            CASE Value 
OF
  SplineMode.DISCRETE_POINTS      : SPLINE_MODE_TO_STRING := StrReplace('DISCRETE_POINTS ({0})'      ,'{0}' , UINT_TO_STRING(Value));
  SplineMode.BEZIER_SPLINE        : SPLINE_MODE_TO_STRING := StrReplace('BEZIER_SPLINE ({0})'        ,'{0}' , UINT_TO_STRING(Value));
  SplineMode.B_SPLINES            : SPLINE_MODE_TO_STRING := StrReplace('B_SPLINES ({0})'            ,'{0}' , UINT_TO_STRING(Value));
  SplineMode.CUBIC_HERMITE_SPLINE : SPLINE_MODE_TO_STRING := StrReplace('CUBIC_HERMITE_SPLINE ({0})' ,'{0}' , UINT_TO_STRING(Value));
  SplineMode.C_SPLINES            : SPLINE_MODE_TO_STRING := StrReplace('C_SPLINES ({0})'            ,'{0}' , UINT_TO_STRING(Value));
ELSE
  SPLINE_MODE_TO_STRING := CONCAT('SPLINE_MODE_TO_STRING Function: Error -> no parsing for value ', UINT_TO_STRING(Value));
END_CASE
          
END_FUNCTION

FUNCTION STEP_MODE_TO_STRING : STRING
// ------------------------------------------------------------------------- 
//  SRCI Robot Library                                                
// ------------------------------------------------------------------------- 
//                                                                           
//  Object:      STEP_MODE_TO_STRING                                       
//  Author:      Thorsten Brach                                                
//  Date:        2025-01-18
//
//  Description:                                              
//   
//                                                                           
//  Copyright: 
//    (C) 2025 Thorsten Brach. All rights reserved                                                                                                                                            
//             Licensed under the MIT License.
//                                                                           
//  Disclaimer:                                                                           
//    This project is provided without any guarantee and can be used for   
//    private and commercial purposes. Any use is at the user’s 
//    own risk and responsibility.
//
// -------------------------------------------------------------------------
VAR_INPUT
  /// StepMode
  Value : StepMode;
END_VAR

            CASE Value 
OF  
  StepMode.DEACTIVATE : STEP_MODE_TO_STRING := StrReplace('DEACTIVATE ({0})' ,'{0}' , USINT_TO_STRING(Value));
  StepMode.BLENDING   : STEP_MODE_TO_STRING := StrReplace('BLENDING ({0})'   ,'{0}' , USINT_TO_STRING(Value));
  StepMode.EXACT_STOP : STEP_MODE_TO_STRING := StrReplace('EXACT_STOP ({0})' ,'{0}' , USINT_TO_STRING(Value));
ELSE
  STEP_MODE_TO_STRING := CONCAT('STEP_MODE_TO_STRING Function: Error -> no parsing for value ', USINT_TO_STRING(Value));
END_CASE
          
END_FUNCTION

FUNCTION STOP_MODE_TO_STRING : STRING
// ------------------------------------------------------------------------- 
//  SRCI Robot Library                                                
// ------------------------------------------------------------------------- 
//                                                                           
//  Object:      STOP_MODE_TO_STRING                                       
//  Author:      Thorsten Brach                                                
//  Date:        2025-01-24
//
//  Description:                                              
//   
//                                                                           
//  Copyright: 
//    (C) 2025 Thorsten Brach. All rights reserved                                                                                                                                            
//             Licensed under the MIT License.
//                                                                           
//  Disclaimer:                                                                           
//    This project is provided without any guarantee and can be used for   
//    private and commercial purposes. Any use is at the user’s 
//    own risk and responsibility.
//
// -------------------------------------------------------------------------
VAR_INPUT
  /// StopMode
  Value : StopMode;
END_VAR

            CASE Value 
OF
  StopMode.STOP_ALL_SUBPROGRAMS : STOP_MODE_TO_STRING := StrReplace('STOP_ALL_SUBPROGRAMS ({0})','{0}' , USINT_TO_STRING(Value));
  StopMode.STOP_INSTANCE_ID     : STOP_MODE_TO_STRING := StrReplace('STOP_INSTANCE_ID ({0})'    ,'{0}' , USINT_TO_STRING(Value));
  StopMode.STOP_JOB_ID          : STOP_MODE_TO_STRING := StrReplace('STOP_JOB_ID ({0})'         ,'{0}' , USINT_TO_STRING(Value));
ELSE
  STOP_MODE_TO_STRING := CONCAT('STOP_MODE_TO_STRING Function: Error -> no parsing for value ', USINT_TO_STRING(Value));
END_CASE
          
END_FUNCTION

FUNCTION SYNC_IN_MODE_TO_STRING : STRING
// ------------------------------------------------------------------------- 
//  SRCI Robot Library                                                
// ------------------------------------------------------------------------- 
//                                                                           
//  Object:      SYNC_IN_MODE_TO_STRING                                       
//  Author:      Thorsten Brach                                                
//  Date:        2025-02-01
//
//  Description:                                              
//   
//                                                                           
//  Copyright: 
//    (C) 2025 Thorsten Brach. All rights reserved                                                                                                                                            
//             Licensed under the MIT License.
//                                                                           
//  Disclaimer:                                                                           
//    This project is provided without any guarantee and can be used for   
//    private and commercial purposes. Any use is at the user’s 
//    own risk and responsibility.
//
// -------------------------------------------------------------------------
VAR_INPUT
  /// SyncInMode
  Value : SyncInMode;
END_VAR

            CASE Value 
OF
  SyncInMode.IN_SYNC_IN_ZONE : SYNC_IN_MODE_TO_STRING := StrReplace('IN_SYNC_IN_ZONE ({0})','{0}' , USINT_TO_STRING(Value));
  SyncInMode.AFTER_DISTANCE  : SYNC_IN_MODE_TO_STRING := StrReplace('AFTER_DISTANCE ({0})' ,'{0}' , USINT_TO_STRING(Value));
  SyncInMode.AFTER_TIME      : SYNC_IN_MODE_TO_STRING := StrReplace('AFTER_TIME ({0})'     ,'{0}' , USINT_TO_STRING(Value));
  SyncInMode.IMMEDIATELY     : SYNC_IN_MODE_TO_STRING := StrReplace('IMMEDIATELY ({0})'    ,'{0}' , USINT_TO_STRING(Value));
ELSE
  SYNC_IN_MODE_TO_STRING := CONCAT('SYNC_IN_MODE_TO_STRING Function: Error -> no parsing for value ', USINT_TO_STRING(Value));
END_CASE
          
END_FUNCTION

FUNCTION SYNC_MODE_TO_STRING : STRING
// ------------------------------------------------------------------------- 
//  SRCI Robot Library                                                
// ------------------------------------------------------------------------- 
//                                                                           
//  Object:      SYNC_MODE_TO_STRING                                       
//  Author:      Thorsten Brach                                                
//  Date:        2025-02-23
//
//  Description:                                              
//   
//                                                                           
//  Copyright: 
//    (C) 2025 Thorsten Brach. All rights reserved                                                                                                                                            
//             Licensed under the MIT License.
//                                                                           
//  Disclaimer:                                                                           
//    This project is provided without any guarantee and can be used for   
//    private and commercial purposes. Any use is at the user’s 
//    own risk and responsibility.
//
// -------------------------------------------------------------------------
VAR_INPUT
  /// SyncMode
  Value : SyncMode;
END_VAR

            CASE Value 
OF
  SyncMode.NO_SYNCHRONIZATION : SYNC_MODE_TO_STRING := StrReplace('NO_SYNCHRONIZATION ({0})','{0}' , USINT_TO_STRING(Value));
  SyncMode.CLIENT_TO_SERVER   : SYNC_MODE_TO_STRING := StrReplace('CLIENT_TO_SERVER ({0})'  ,'{0}' , USINT_TO_STRING(Value));
  SyncMode.SERVER_TO_CLIENT   : SYNC_MODE_TO_STRING := StrReplace('SERVER_TO_CLIENT ({0})'  ,'{0}' , USINT_TO_STRING(Value));
  SyncMode.AUTOMATIC          : SYNC_MODE_TO_STRING := StrReplace('AUTOMATIC ({0})'         ,'{0}' , USINT_TO_STRING(Value));
ELSE
  SYNC_MODE_TO_STRING := CONCAT('SYNC_MODE_TO_STRING Function: Error -> no parsing for value ', USINT_TO_STRING(Value));
END_CASE
          
END_FUNCTION

FUNCTION SYNC_REACTION_TO_STRING : STRING
// ------------------------------------------------------------------------- 
//  SRCI Robot Library                                                
// ------------------------------------------------------------------------- 
//                                                                           
//  Object:      SYNC_REACTION_TO_STRING                                       
//  Author:      Thorsten Brach                                                
//  Date:        2025-01-24
//
//  Description:                                              
//   
//                                                                           
//  Copyright: 
//    (C) 2025 Thorsten Brach. All rights reserved                                                                                                                                            
//             Licensed under the MIT License.
//                                                                           
//  Disclaimer:                                                                           
//    This project is provided without any guarantee and can be used for   
//    private and commercial purposes. Any use is at the user’s 
//    own risk and responsibility.
//
// -------------------------------------------------------------------------
VAR_INPUT
  /// SyncReaction
  Value : SyncReaction;
END_VAR

            CASE Value 
OF
  SyncReaction.NO_REACTION                      : SYNC_REACTION_TO_STRING := StrReplace('NO_REACTION ({0})'                      ,'{0}' , USINT_TO_STRING(Value));
  SyncReaction.NO_AUTOMATIC_DISABLE             : SYNC_REACTION_TO_STRING := StrReplace('NO_AUTOMATIC_DISABLE ({0})'             ,'{0}' , USINT_TO_STRING(Value));
  SyncReaction.INTERRUPT_WHEN_SEQUENCE_IS_EMPTY : SYNC_REACTION_TO_STRING := StrReplace('INTERRUPT_WHEN_SEQUENCE_IS_EMPTY ({0})' ,'{0}' , USINT_TO_STRING(Value));
  SyncReaction.IMMEDIATE_INTERRUPT              : SYNC_REACTION_TO_STRING := StrReplace('IMMEDIATE_INTERRUPT ({0})'              ,'{0}' , USINT_TO_STRING(Value));
ELSE
  SYNC_REACTION_TO_STRING := CONCAT('SYNC_REACTION_TO_STRING Function: Error -> no parsing for value ', USINT_TO_STRING(Value));
END_CASE
          
END_FUNCTION

FUNCTION SYNC_TIME_TO_STRING : STRING
// ------------------------------------------------------------------------- 
//  SRCI Robot Library                                                
// ------------------------------------------------------------------------- 
//                                                                           
//  Object:      SYNC_TIME_TO_STRING                                       
//  Author:      Thorsten Brach                                                
//  Date:        2025-04-13
//
//  Description:                                              
//   
//                                                                           
//  Copyright: 
//    (C) 2025 Thorsten Brach. All rights reserved                                                                                                                                            
//             Licensed under the MIT License.
//                                                                           
//  Disclaimer:                                                                           
//    This project is provided without any guarantee and can be used for   
//    private and commercial purposes. Any use is at the user’s 
//    own risk and responsibility.
//
// -------------------------------------------------------------------------
VAR_INPUT
  /// SyncTime
  Value : SyncTime;
END_VAR

            CASE Value 
OF
  SyncTime.DURING_START_UP : SYNC_TIME_TO_STRING := StrReplace('DURING_START_UP ({0})','{0}' , DINT_TO_STRING(Value));
  SyncTime.AFTER_START_UP  : SYNC_TIME_TO_STRING := StrReplace('AFTER_START_UP ({0})' ,'{0}' , DINT_TO_STRING(Value));
ELSE
  SYNC_TIME_TO_STRING := CONCAT('SYNC_TIME_TO_STRING Function: Error -> no parsing for value ', DINT_TO_STRING(Value));
END_CASE
          
END_FUNCTION

FUNCTION TELEGRAM_CONTROL_TO_STRING : STRING
// ------------------------------------------------------------------------- 
//  SRCI Robot Library                                                
// ------------------------------------------------------------------------- 
//                                                                           
//  Object:      TELEGRAM_CONTROL_TO_STRING                                       
//  Author:      Thorsten Brach                                                
//  Date:        2024-11-16
//
//  Description:                                              
//   
//                                                                           
//  Copyright: 
//    (C) 2024 Thorsten Brach. All rights reserved                                                                                                                                            
//             Licensed under the MIT License.
//                                                                           
//  Disclaimer:                                                                           
//    This project is provided without any guarantee and can be used for   
//    private and commercial purposes. Any use is at the user’s 
//    own risk and responsibility.
//
// -------------------------------------------------------------------------
VAR_INPUT
  /// Telegram state
  Control : ControlHalfByte;
END_VAR

            CASE Control 
OF
  ControlHalfByte.NONE         : TELEGRAM_CONTROL_TO_STRING := StrReplace('NONE ({0})'        ,'{0}', USINT_TO_STRING(Control));
  ControlHalfByte.INITIALIZE   : TELEGRAM_CONTROL_TO_STRING := StrReplace('INITIALIZE ({0})'  ,'{0}', USINT_TO_STRING(Control));
  ControlHalfByte.RESUME       : TELEGRAM_CONTROL_TO_STRING := StrReplace('RESUME ({0})'      ,'{0}', USINT_TO_STRING(Control));
  ControlHalfByte.RESET        : TELEGRAM_CONTROL_TO_STRING := StrReplace('RESET ({0})'       ,'{0}', USINT_TO_STRING(Control));
  ControlHalfByte.ACK_ERROR    : TELEGRAM_CONTROL_TO_STRING := StrReplace('ACK_ERROR ({0})'   ,'{0}', USINT_TO_STRING(Control));
  ControlHalfByte.CLIENT_ERROR : TELEGRAM_CONTROL_TO_STRING := StrReplace('CLIENT_ERROR ({0})','{0}', USINT_TO_STRING(Control));  
ELSE
  TELEGRAM_CONTROL_TO_STRING := CONCAT('TelegramControlToString-Function: Error -> no parsing for value ', USINT_TO_STRING(Control));
END_CASE 
          
END_FUNCTION

FUNCTION TELEGRAM_STATE_TO_STRING : STRING
// ------------------------------------------------------------------------- 
//  SRCI Robot Library                                                
// ------------------------------------------------------------------------- 
//                                                                           
//  Object:      TelegramStateToString                                       
//  Author:      Thorsten Brach                                                
//  Date:        2024-11-16
//
//  Description:                                              
//   
//                                                                           
//  Copyright: 
//    (C) 2024 Thorsten Brach. All rights reserved                                                                                                                                            
//             Licensed under the MIT License.
//                                                                           
//  Disclaimer:                                                                           
//    This project is provided without any guarantee and can be used for   
//    private and commercial purposes. Any use is at the user’s 
//    own risk and responsibility.
//
// -------------------------------------------------------------------------
VAR_INPUT
  /// Telegram state
  State : TelegramState;
END_VAR

            CASE State 
OF
  TelegramState.UNDEFINED                                          : TELEGRAM_STATE_TO_STRING := StrReplace('UNDEFINED ({0})'                                          ,'{0}', USINT_TO_STRING(State));
  TelegramState.ERROR_161_TELEGRAM_CONTROL_MISMATCH_TELEGRAM_STATE : TELEGRAM_STATE_TO_STRING := StrReplace('ERROR_161_TELEGRAM_CONTROL_MISMATCH_TELEGRAM_STATE ({0})' ,'{0}', USINT_TO_STRING(State));
  TelegramState.ERROR_162_INIT_LOST_UNKNOWN                        : TELEGRAM_STATE_TO_STRING := StrReplace('ERROR_162_INIT_LOST_UNKNOWN ({0})'                        ,'{0}', USINT_TO_STRING(State));
  TelegramState.ERROR_163_TELEGRAM_LENGTH_MISMATCH                 : TELEGRAM_STATE_TO_STRING := StrReplace('ERROR_163_TELEGRAM_LENGTH_MISMATCH ({0})'                 ,'{0}', USINT_TO_STRING(State));
  TelegramState.ERROR_164_SRCI_MAJOR_VERSION_INCOMPATIBLE          : TELEGRAM_STATE_TO_STRING := StrReplace('ERROR_164_SRCI_MAJOR_VERSION_INCOMPATIBLE ({0})'          ,'{0}', USINT_TO_STRING(State));
  TelegramState.ERROR_165_LIFESIGN_TIMEOUT                         : TELEGRAM_STATE_TO_STRING := StrReplace('ERROR_165_LIFESIGN_TIMEOUT ({0})'                         ,'{0}', USINT_TO_STRING(State));
  TelegramState.ERROR_166_CYCLIC_DATA_TOO_LARGE                    : TELEGRAM_STATE_TO_STRING := StrReplace('ERROR_166_CYCLIC_DATA_TOO_LARGE ({0})'                    ,'{0}', USINT_TO_STRING(State));
  TelegramState.ERROR_167_INTERFACE_WAS_RESET_AFTER_INIT           : TELEGRAM_STATE_TO_STRING := StrReplace('ERROR_167_INTERFACE_WAS_RESET_AFTER_INIT ({0})'           ,'{0}', USINT_TO_STRING(State));
  TelegramState.ERROR_168_TELEGRAM_SEQ_TIMEOUT                     : TELEGRAM_STATE_TO_STRING := StrReplace('ERROR_168_TELEGRAM_SEQ_TIMEOUT ({0})'                     ,'{0}', USINT_TO_STRING(State));
  TelegramState.ERROR_169_TELEGRAM_NO_CHANGED_AFTER_INIT           : TELEGRAM_STATE_TO_STRING := StrReplace('ERROR_169_TELEGRAM_NO_CHANGED_AFTER_INIT ({0})'           ,'{0}', USINT_TO_STRING(State));
  TelegramState.ERROR_170_AXESGROUP_ID_INVALID                     : TELEGRAM_STATE_TO_STRING := StrReplace('ERROR_170_AXESGROUP_ID_INVALID ({0})'                     ,'{0}', USINT_TO_STRING(State));
  TelegramState.ERROR_171_TELEGRAM_NUMBER_INVALID                  : TELEGRAM_STATE_TO_STRING := StrReplace('ERROR_171_TELEGRAM_NUMBER_INVALID ({0})'                  ,'{0}', USINT_TO_STRING(State));
  TelegramState.ERROR_172_TELEGRAM_NUMBER_NOT_SUPPORTED            : TELEGRAM_STATE_TO_STRING := StrReplace('ERROR_172_TELEGRAM_NUMBER_NOT_SUPPORTED ({0})'            ,'{0}', USINT_TO_STRING(State));
  TelegramState.ERROR_173_SERVER_CONNECTION_LOST                   : TELEGRAM_STATE_TO_STRING := StrReplace('ERROR_173_SERVER_CONNECTION_LOST ({0})'                   ,'{0}', USINT_TO_STRING(State));
  TelegramState.READY_TO_RESUME                                    : TELEGRAM_STATE_TO_STRING := StrReplace('READY_TO_RESUME ({0})'                                    ,'{0}', USINT_TO_STRING(State));
  TelegramState.READY_FOR_INITIALIZATION                           : TELEGRAM_STATE_TO_STRING := StrReplace('READY_FOR_INITIALIZATION ({0})'                           ,'{0}', USINT_TO_STRING(State));
  TelegramState.INITIALIZED                                        : TELEGRAM_STATE_TO_STRING := StrReplace('INITIALIZED ({0})'                                        ,'{0}', USINT_TO_STRING(State));  
ELSE
  TELEGRAM_STATE_TO_STRING := CONCAT('TELEGRAM_STATE_TO_STRING Function: Error -> no parsing for value ', USINT_TO_STRING(State));
END_CASE 
          
END_FUNCTION

FUNCTION THRESHOLD_MODE_TO_STRING : STRING
// ------------------------------------------------------------------------- 
//  SRCI Robot Library                                                
// ------------------------------------------------------------------------- 
//                                                                           
//  Object:      THRESHOLD_MODE_TO_STRING                                       
//  Author:      Thorsten Brach                                                
//  Date:        2025-01-24
//
//  Description:                                              
//   
//                                                                           
//  Copyright: 
//    (C) 2025 Thorsten Brach. All rights reserved                                                                                                                                            
//             Licensed under the MIT License.
//                                                                           
//  Disclaimer:                                                                           
//    This project is provided without any guarantee and can be used for   
//    private and commercial purposes. Any use is at the user’s 
//    own risk and responsibility.
//
// -------------------------------------------------------------------------
VAR_INPUT
  /// ThresholdMode
  Value : ThresholdMode;
END_VAR

            CASE Value 
OF
  ThresholdMode.AUTOMATIC : THRESHOLD_MODE_TO_STRING := StrReplace('AUTOMATIC ({0})','{0}' , USINT_TO_STRING(Value));
  ThresholdMode.MANUAL    : THRESHOLD_MODE_TO_STRING := StrReplace('MANUAL ({0})'   ,'{0}' , USINT_TO_STRING(Value));
ELSE
  THRESHOLD_MODE_TO_STRING := CONCAT('THRESHOLD_MODE_TO_STRING Function: Error -> no parsing for value ', USINT_TO_STRING(Value));
END_CASE
          
END_FUNCTION

FUNCTION TOOL_CALCULATION_MODE_TO_STRING : STRING
// ------------------------------------------------------------------------- 
//  SRCI Robot Library                                                
// ------------------------------------------------------------------------- 
//                                                                           
//  Object:      TOOL_CALCULATION_MODE_TO_STRING                                       
//  Author:      Thorsten Brach                                                
//  Date:        2025-02-01
//
//  Description:                                              
//   
//                                                                           
//  Copyright: 
//    (C) 2025 Thorsten Brach. All rights reserved                                                                                                                                            
//             Licensed under the MIT License.
//                                                                           
//  Disclaimer:                                                                           
//    This project is provided without any guarantee and can be used for   
//    private and commercial purposes. Any use is at the user’s 
//    own risk and responsibility.
//
// -------------------------------------------------------------------------
VAR_INPUT
  /// ToolCalculationMode
  Value : ToolCalculationMode;
END_VAR

            CASE Value 
OF
  ToolCalculationMode.TWO_POINT_Z_METHOD   : TOOL_CALCULATION_MODE_TO_STRING := StrReplace('TWO_POINT_Z_METHOD ({0})'  ,'{0}' , SINT_TO_STRING(Value));
  ToolCalculationMode.THREE_POINT_METHOD   : TOOL_CALCULATION_MODE_TO_STRING := StrReplace('THREE_POINT_METHOD ({0})'  ,'{0}' , SINT_TO_STRING(Value));
  ToolCalculationMode.FOUR_POINT_METHOD    : TOOL_CALCULATION_MODE_TO_STRING := StrReplace('FOUR_POINT_METHOD ({0})'   ,'{0}' , SINT_TO_STRING(Value));
  ToolCalculationMode.FIVE_POINT_METHOD    : TOOL_CALCULATION_MODE_TO_STRING := StrReplace('FIVE_POINT_METHOD ({0})'   ,'{0}' , SINT_TO_STRING(Value));
  ToolCalculationMode.SIX_POINT_METHOD     : TOOL_CALCULATION_MODE_TO_STRING := StrReplace('SIX_POINT_METHOD ({0})'    ,'{0}' , SINT_TO_STRING(Value));
  ToolCalculationMode.ABC_WORLD_METHOD     : TOOL_CALCULATION_MODE_TO_STRING := StrReplace('ABC_WORLD_METHOD ({0})'    ,'{0}' , SINT_TO_STRING(Value));
  ToolCalculationMode.ABC_TWO_POINT_METHOD : TOOL_CALCULATION_MODE_TO_STRING := StrReplace('ABC_TWO_POINT_METHOD ({0})','{0}' , SINT_TO_STRING(Value));
ELSE
  TOOL_CALCULATION_MODE_TO_STRING := CONCAT('TOOL_CALCULATION_MODE_TO_STRING Function: Error -> no parsing for value ', SINT_TO_STRING(Value));
END_CASE
          
END_FUNCTION

FUNCTION TRAJECTORY_MODE_TO_STRING : STRING
// ------------------------------------------------------------------------- 
//  SRCI Robot Library                                                
// ------------------------------------------------------------------------- 
//                                                                           
//  Object:      TRAJECTORY_MODE_TO_STRING                                       
//  Author:      Thorsten Brach                                                
//  Date:        2025-03-01
//
//  Description:                                              
//   
//                                                                           
//  Copyright: 
//    (C) 2025 Thorsten Brach. All rights reserved                                                                                                                                            
//             Licensed under the MIT License.
//                                                                           
//  Disclaimer:                                                                           
//    This project is provided without any guarantee and can be used for   
//    private and commercial purposes. Any use is at the user’s 
//    own risk and responsibility.
//
// -------------------------------------------------------------------------
VAR_INPUT
  /// TrajectoryMode
  Value : TrajectoryMode;
END_VAR

            CASE Value 
OF
  TrajectoryMode.INVALID          : TRAJECTORY_MODE_TO_STRING := StrReplace('INVALID ({0})'         ,'{0}' , USINT_TO_STRING(Value));
  TrajectoryMode.LINEAR_MOVEMENT  : TRAJECTORY_MODE_TO_STRING := StrReplace('LINEAR_MOVEMENT ({0})' ,'{0}' , USINT_TO_STRING(Value));
  TrajectoryMode.PTP_MOVEMENT     : TRAJECTORY_MODE_TO_STRING := StrReplace('PTP_MOVEMENT ({0})'    ,'{0}' , USINT_TO_STRING(Value));
ELSE
  TRAJECTORY_MODE_TO_STRING := CONCAT('TRAJECTORY_MODE_TO_STRING Function: Error -> no parsing for value ', USINT_TO_STRING(Value));
END_CASE
          
END_FUNCTION

FUNCTION TRANSFORM_MODE_TO_STRING : STRING
// ------------------------------------------------------------------------- 
//  SRCI Robot Library                                                
// ------------------------------------------------------------------------- 
//                                                                           
//  Object:      TRANSFORM_MODE_TO_STRING                                       
//  Author:      Thorsten Brach                                                
//  Date:        2025-01-24
//
//  Description:                                              
//   
//                                                                           
//  Copyright: 
//    (C) 2025 Thorsten Brach. All rights reserved                                                                                                                                            
//             Licensed under the MIT License.
//                                                                           
//  Disclaimer:                                                                           
//    This project is provided without any guarantee and can be used for   
//    private and commercial purposes. Any use is at the user’s 
//    own risk and responsibility.
//
// -------------------------------------------------------------------------
VAR_INPUT
  /// TransformMode
  Value : TransformMode;
END_VAR

            CASE Value 
OF
  TransformMode.MIRROR_AT_POINT             : TRANSFORM_MODE_TO_STRING := StrReplace('MIRROR_AT_POINT ({0})'             ,'{0}' , SINT_TO_STRING(Value));
  TransformMode.MIRROR_AT_STRAIGHT_LINE     : TRANSFORM_MODE_TO_STRING := StrReplace('MIRROR_AT_STRAIGHT_LINE ({0})'     ,'{0}' , SINT_TO_STRING(Value));
  TransformMode.MIRROR_AT_PLANE             : TRANSFORM_MODE_TO_STRING := StrReplace('MIRROR_AT_PLANE ({0})'             ,'{0}' , SINT_TO_STRING(Value));
  TransformMode.ROTATE_AROUND_STRAIGHT_LINE : TRANSFORM_MODE_TO_STRING := StrReplace('ROTATE_AROUND_STRAIGHT_LINE ({0})' ,'{0}' , SINT_TO_STRING(Value));
  TransformMode.SHIFT_BY_VECTOR             : TRANSFORM_MODE_TO_STRING := StrReplace('SHIFT_BY_VECTOR ({0})'             ,'{0}' , SINT_TO_STRING(Value));
ELSE
  TRANSFORM_MODE_TO_STRING := CONCAT('TRANSFORM_MODE_TO_STRING Function: Error -> no parsing for value ', SINT_TO_STRING(Value));
END_CASE
          
END_FUNCTION

FUNCTION TRIGGER_CONDITION_TO_STRING : STRING
// ------------------------------------------------------------------------- 
//  SRCI Robot Library                                                
// ------------------------------------------------------------------------- 
//                                                                           
//  Object:      TRIGGER_CONDITION_TO_STRING                                       
//  Author:      Thorsten Brach                                                
//  Date:        2025-02-01
//
//  Description:                                              
//   
//                                                                           
//  Copyright: 
//    (C) 2025 Thorsten Brach. All rights reserved                                                                                                                                            
//             Licensed under the MIT License.
//                                                                           
//  Disclaimer:                                                                           
//    This project is provided without any guarantee and can be used for   
//    private and commercial purposes. Any use is at the user’s 
//    own risk and responsibility.
//
// -------------------------------------------------------------------------
VAR_INPUT
  /// TriggerCondition
  Value : TriggerCondition;
END_VAR

            CASE Value 
OF
  TriggerCondition.TARGET_POSITION_TIME_MS                : TRIGGER_CONDITION_TO_STRING := StrReplace('TARGET_POSITION_TIME_MS ({0})'               ,'{0}' , SINT_TO_STRING(Value));
  TriggerCondition.TARGET_POSITION_TCP_VELOCITY_ABSOLUTE  : TRIGGER_CONDITION_TO_STRING := StrReplace('TARGET_POSITION_TCP_VELOCITY_ABSOLUTE ({0})' ,'{0}' , SINT_TO_STRING(Value));
  TriggerCondition.TARGET_POSITION_TCP_VELOCITY_PERCENT   : TRIGGER_CONDITION_TO_STRING := StrReplace('TARGET_POSITION_TCP_VELOCITY_PERCENT ({0})'  ,'{0}' , SINT_TO_STRING(Value));
  TriggerCondition.TARGET_POSITION_DISTANCE_ABSOLUTE      : TRIGGER_CONDITION_TO_STRING := StrReplace('TARGET_POSITION_DISTANCE_ABSOLUTE ({0})'     ,'{0}' , SINT_TO_STRING(Value));
  TriggerCondition.TARGET_POSITION_DISTANCE_PERCENT       : TRIGGER_CONDITION_TO_STRING := StrReplace('TARGET_POSITION_DISTANCE_PERCENT ({0})'      ,'{0}' , SINT_TO_STRING(Value));
  TriggerCondition.UNDEFINED                              : TRIGGER_CONDITION_TO_STRING := StrReplace('UNDEFINED ({0})'                             ,'{0}' , SINT_TO_STRING(Value));
  TriggerCondition.START_POSITION_DISTANCE_PERCENT        : TRIGGER_CONDITION_TO_STRING := StrReplace('START_POSITION_DISTANCE_PERCENT ({0})'       ,'{0}' , SINT_TO_STRING(Value));
  TriggerCondition.START_POSITION_DISTANCE_ABSOLUTE       : TRIGGER_CONDITION_TO_STRING := StrReplace('START_POSITION_DISTANCE_ABSOLUTE ({0})'      ,'{0}' , SINT_TO_STRING(Value));
  TriggerCondition.START_POSITION_TCP_VELOCITY_PERCENT    : TRIGGER_CONDITION_TO_STRING := StrReplace('START_POSITION_TCP_VELOCITY_PERCENT ({0})'   ,'{0}' , SINT_TO_STRING(Value));
  TriggerCondition.START_POSITION_TCP_VELOCIT_ABSOLUTE    : TRIGGER_CONDITION_TO_STRING := StrReplace('START_POSITION_TCP_VELOCIT_ABSOLUTE ({0})'   ,'{0}' , SINT_TO_STRING(Value));
  TriggerCondition.START_POSITION_TIME_MS                 : TRIGGER_CONDITION_TO_STRING := StrReplace('START_POSITION_TCP_VELOCIT_ABSOLUTE ({0})'   ,'{0}' , SINT_TO_STRING(Value));
ELSE
  TRIGGER_CONDITION_TO_STRING := CONCAT('TRIGGER_CONDITION_TO_STRING Function: Error -> no parsing for value ', SINT_TO_STRING(Value));
END_CASE
          
END_FUNCTION

FUNCTION TRIGGER_MODE_IO_TO_STRING : STRING
// ------------------------------------------------------------------------- 
//  SRCI Robot Library                                                
// ------------------------------------------------------------------------- 
//                                                                           
//  Object:      TRIGGER_MODE_IO_TO_STRING                                       
//  Author:      Thorsten Brach                                                
//  Date:        2025-02-01
//
//  Description:                                              
//   
//                                                                           
//  Copyright: 
//    (C) 2025 Thorsten Brach. All rights reserved                                                                                                                                            
//             Licensed under the MIT License.
//                                                                           
//  Disclaimer:                                                                           
//    This project is provided without any guarantee and can be used for   
//    private and commercial purposes. Any use is at the user’s 
//    own risk and responsibility.
//
// -------------------------------------------------------------------------
VAR_INPUT
  /// TriggerModeIo
  Value : TriggerModeIo;
END_VAR

            CASE Value 
OF
  TriggerModeIo.INVALID                                                             : TRIGGER_MODE_IO_TO_STRING := StrReplace('INVALID ({0})'                                                              ,'{0}' , SINT_TO_STRING(Value));
  TriggerModeIo.DIGITAL_INPUT_RISING_EDGE                                           : TRIGGER_MODE_IO_TO_STRING := StrReplace('DIGITAL_INPUT_RISING_EDGE ({0})'                                            ,'{0}' , SINT_TO_STRING(Value));
  TriggerModeIo.DIGITAL_INPUT_FALLING_EDGE                                          : TRIGGER_MODE_IO_TO_STRING := StrReplace('DIGITAL_INPUT_FALLING_EDGE ({0})'                                           ,'{0}' , SINT_TO_STRING(Value));
  TriggerModeIo.DIGITAL_INPUT_RISING_OR_FALLING_EDGE                                : TRIGGER_MODE_IO_TO_STRING := StrReplace('DIGITAL_INPUT_RISING_OR_FALLING_EDGE ({0})'                                 ,'{0}' , SINT_TO_STRING(Value));
  TriggerModeIo.DIGITAL_INPUT_RISING_OR_FALLING_EDGE_INVERTED                       : TRIGGER_MODE_IO_TO_STRING := StrReplace('DIGITAL_INPUT_RISING_OR_FALLING_EDGE_INVERTED ({0})'                        ,'{0}' , SINT_TO_STRING(Value));
  TriggerModeIo.DIGITAL_OUTPUT_RISING_EDGE                                          : TRIGGER_MODE_IO_TO_STRING := StrReplace('DIGITAL_OUTPUT_RISING_EDGE ({0})'                                           ,'{0}' , SINT_TO_STRING(Value));
  TriggerModeIo.DIGITAL_OUTPUT_FALLING_EDGE                                         : TRIGGER_MODE_IO_TO_STRING := StrReplace('DIGITAL_OUTPUT_FALLING_EDGE ({0})'                                          ,'{0}' , SINT_TO_STRING(Value));
  TriggerModeIo.DIGITAL_OUTPUT_RISING_OR_FALLING_EDGE                               : TRIGGER_MODE_IO_TO_STRING := StrReplace('DIGITAL_OUTPUT_RISING_OR_FALLING_EDGE ({0})'                                ,'{0}' , SINT_TO_STRING(Value));
  TriggerModeIo.DIGITAL_OUTPUT_RISING_OR_FALLING_EDGE_INVERTED                      : TRIGGER_MODE_IO_TO_STRING := StrReplace('DIGITAL_OUTPUT_RISING_OR_FALLING_EDGE_INVERTED ({0})'                       ,'{0}' , SINT_TO_STRING(Value));
  TriggerModeIo.ANALOG_INPUT_EXCEEDING_DEFINED_THRESHOLD                            : TRIGGER_MODE_IO_TO_STRING := StrReplace('ANALOG_INPUT_EXCEEDING_DEFINED_THRESHOLD ({0})'                             ,'{0}' , SINT_TO_STRING(Value));
  TriggerModeIo.ANALOG_INPUT_FALLING_BELOW_DEFINED_THRESHOLD                        : TRIGGER_MODE_IO_TO_STRING := StrReplace('ANALOG_INPUT_FALLING_BELOW_DEFINED_THRESHOLD ({0})'                         ,'{0}' , SINT_TO_STRING(Value));
  TriggerModeIo.ANALOG_INPUT_EXCEEDING_OR_FALLING_BELOW_DEFINED_THRESHOLD           : TRIGGER_MODE_IO_TO_STRING := StrReplace('ANALOG_INPUT_EXCEEDING_OR_FALLING_BELOW_DEFINED_THRESHOLD ({0})'            ,'{0}' , SINT_TO_STRING(Value));
  TriggerModeIo.ANALOG_INPUT_EXCEEDING_OR_FALLING_BELOW_DEFINED_THRESHOLD_INVERTED  : TRIGGER_MODE_IO_TO_STRING := StrReplace('ANALOG_INPUT_EXCEEDING_OR_FALLING_BELOW_DEFINED_THRESHOLD_INVERTED ({0})'   ,'{0}' , SINT_TO_STRING(Value));
  TriggerModeIo.ANALOG_INPUT_ENTERING_DEFINED_RANGE                                 : TRIGGER_MODE_IO_TO_STRING := StrReplace('ANALOG_INPUT_ENTERING_DEFINED_RANGE ({0})'                                  ,'{0}' , SINT_TO_STRING(Value));
  TriggerModeIo.ANALOG_INPUT_LEAVING_DEFINED_RANGE                                  : TRIGGER_MODE_IO_TO_STRING := StrReplace('ANALOG_INPUT_LEAVING_DEFINED_RANGE ({0})'                                   ,'{0}' , SINT_TO_STRING(Value));
  TriggerModeIo.ANALOG_INPUT_ENTERING_OR_LEAVING_DEFINED_RANGE                      : TRIGGER_MODE_IO_TO_STRING := StrReplace('ANALOG_INPUT_ENTERING_OR_LEAVING_DEFINED_RANGE ({0})'                       ,'{0}' , SINT_TO_STRING(Value));
  TriggerModeIo.ANALOG_INPUT_ENTERING_OR_LEAVING_DEFINED_RANGE_INVERTED             : TRIGGER_MODE_IO_TO_STRING := StrReplace('ANALOG_INPUT_ENTERING_OR_LEAVING_DEFINED_RANGE_INVERTED ({0})'              ,'{0}' , SINT_TO_STRING(Value));
  TriggerModeIo.ANALOG_OUTPUT_EXCEEDING_DEFINED_THRESHOLD                           : TRIGGER_MODE_IO_TO_STRING := StrReplace('ANALOG_OUTPUT_EXCEEDING_DEFINED_THRESHOLD ({0})'                            ,'{0}' , SINT_TO_STRING(Value));
  TriggerModeIo.ANALOG_OUTPUT_FALLING_BELOW_DEFINED_THRESHOLD                       : TRIGGER_MODE_IO_TO_STRING := StrReplace('ANALOG_OUTPUT_FALLING_BELOW_DEFINED_THRESHOLD ({0})'                        ,'{0}' , SINT_TO_STRING(Value));
  TriggerModeIo.ANALOG_OUTPUT_EXCEEDING_OR_FALLING_BELOW_DEFINED_THRESHOLD          : TRIGGER_MODE_IO_TO_STRING := StrReplace('ANALOG_OUTPUT_EXCEEDING_OR_FALLING_BELOW_DEFINED_THRESHOLD ({0})'           ,'{0}' , SINT_TO_STRING(Value));
  TriggerModeIo.ANALOG_OUTPUT_EXCEEDING_OR_FALLING_BELOW_DEFINED_THRESHOLD_INVERTED : TRIGGER_MODE_IO_TO_STRING := StrReplace('ANALOG_OUTPUT_EXCEEDING_OR_FALLING_BELOW_DEFINED_THRESHOLD_INVERTED ({0})'  ,'{0}' , SINT_TO_STRING(Value));
  TriggerModeIo.ANALOG_OUTPUT_ENTERING_DEFINED_RANGE                                : TRIGGER_MODE_IO_TO_STRING := StrReplace('ANALOG_OUTPUT_ENTERING_DEFINED_RANGE ({0})'                                 ,'{0}' , SINT_TO_STRING(Value));
  TriggerModeIo.ANALOG_OUTPUT_LEAVING_DEFINED_RANGE                                 : TRIGGER_MODE_IO_TO_STRING := StrReplace('ANALOG_OUTPUT_LEAVING_DEFINED_RANGE ({0})'                                  ,'{0}' , SINT_TO_STRING(Value));
  TriggerModeIo.ANALOG_OUTPUT_ENTERING_OR_LEAVING_DEFINED_RANGE                     : TRIGGER_MODE_IO_TO_STRING := StrReplace('ANALOG_OUTPUT_ENTERING_OR_LEAVING_DEFINED_RANGE ({0})'                      ,'{0}' , SINT_TO_STRING(Value));
  TriggerModeIo.ANALOG_OUTPUT_ENTERING_OR_LEAVING_DEFINED_RANGE_INVERTED            : TRIGGER_MODE_IO_TO_STRING := StrReplace('ANALOG_OUTPUT_ENTERING_OR_LEAVING_DEFINED_RANGE_INVERTED ({0})'             ,'{0}' , SINT_TO_STRING(Value));
  TriggerModeIo.INTEGER_REGISTER_EXCEEDING_DEFINED_THRESHOLD                        : TRIGGER_MODE_IO_TO_STRING := StrReplace('INTEGER_REGISTER_EXCEEDING_DEFINED_THRESHOLD ({0})'                         ,'{0}' , SINT_TO_STRING(Value));
  TriggerModeIo.INTEGER_REGISTER_FALLING_BELOW_DEFINED_THRESHOLD                    : TRIGGER_MODE_IO_TO_STRING := StrReplace('INTEGER_REGISTER_FALLING_BELOW_DEFINED_THRESHOLD ({0})'                     ,'{0}' , SINT_TO_STRING(Value));
  TriggerModeIo.INTEGER_REGISTER_EXCEEDING_OR_FALLING_BELOW_DEFINED_THRESHOLD       : TRIGGER_MODE_IO_TO_STRING := StrReplace('INTEGER_REGISTER_EXCEEDING_OR_FALLING_BELOW_DEFINED_THRESHOLD ({0})'        ,'{0}' , SINT_TO_STRING(Value));
  TriggerModeIo.INTEGER_REGISTER_EXCEEDING_OR_FALLING_BELOW_DEFINED_VALUE_INVERTED  : TRIGGER_MODE_IO_TO_STRING := StrReplace('INTEGER_REGISTER_EXCEEDING_OR_FALLING_BELOW_DEFINED_VALUE_INVERTED ({0})'   ,'{0}' , SINT_TO_STRING(Value));
  TriggerModeIo.INTEGER_REGISTER_ENTERING_DEFINED_RANGE                             : TRIGGER_MODE_IO_TO_STRING := StrReplace('INTEGER_REGISTER_ENTERING_DEFINED_RANGE ({0})'                              ,'{0}' , SINT_TO_STRING(Value));
  TriggerModeIo.INTEGER_REGISTER_LEAVING_DEFINED_RANGE                              : TRIGGER_MODE_IO_TO_STRING := StrReplace('INTEGER_REGISTER_LEAVING_DEFINED_RANGE ({0})'                               ,'{0}' , SINT_TO_STRING(Value));
  TriggerModeIo.INTEGER_REGISTER_ENTERING_OR_LEAVING_DEFINED_RANGE                  : TRIGGER_MODE_IO_TO_STRING := StrReplace('INTEGER_REGISTER_ENTERING_OR_LEAVING_DEFINED_RANGE ({0})'                   ,'{0}' , SINT_TO_STRING(Value));
  TriggerModeIo.INTEGER_REGISTER_ENTERING_OR_LEAVING_DEFINED_RANGE_INVERTED         : TRIGGER_MODE_IO_TO_STRING := StrReplace('INTEGER_REGISTER_ENTERING_OR_LEAVING_DEFINED_RANGE_INVERTED ({0})'          ,'{0}' , SINT_TO_STRING(Value));
  TriggerModeIo.REAL_REGISTER_EXCEEDING_DEFINED_THRESHOLD                           : TRIGGER_MODE_IO_TO_STRING := StrReplace('REAL_REGISTER_EXCEEDING_DEFINED_THRESHOLD ({0})'                            ,'{0}' , SINT_TO_STRING(Value));
  TriggerModeIo.REAL_REGISTER_FALLING_BELOW_DEFINED_THRESHOLD                       : TRIGGER_MODE_IO_TO_STRING := StrReplace('REAL_REGISTER_FALLING_BELOW_DEFINED_THRESHOLD ({0})'                        ,'{0}' , SINT_TO_STRING(Value));
  TriggerModeIo.REAL_REGISTER_EXCEEDING_OR_FALLING_BELOW_DEFINED_THRESHOLD          : TRIGGER_MODE_IO_TO_STRING := StrReplace('REAL_REGISTER_EXCEEDING_OR_FALLING_BELOW_DEFINED_THRESHOLD ({0})'           ,'{0}' , SINT_TO_STRING(Value));
  TriggerModeIo.REAL_REGISTER_EXCEEDING_OR_FALLING_BELOW_DEFINED_THRESHOLD_INVERTED : TRIGGER_MODE_IO_TO_STRING := StrReplace('REAL_REGISTER_EXCEEDING_OR_FALLING_BELOW_DEFINED_THRESHOLD_INVERTED ({0})'  ,'{0}' , SINT_TO_STRING(Value));
  TriggerModeIo.REAL_REGISTER_ENTERING_DEFINED_RANGE                                : TRIGGER_MODE_IO_TO_STRING := StrReplace('REAL_REGISTER_ENTERING_DEFINED_RANGE ({0})'                                 ,'{0}' , SINT_TO_STRING(Value));
  TriggerModeIo.REAL_REGISTER_LEAVING_DEFINED_RANGE                                 : TRIGGER_MODE_IO_TO_STRING := StrReplace('REAL_REGISTER_LEAVING_DEFINED_RANGE ({0})'                                  ,'{0}' , SINT_TO_STRING(Value));
  TriggerModeIo.REAL_REGISTER_ENTERING_OR_LEAVING_DEFINED_RANGE                     : TRIGGER_MODE_IO_TO_STRING := StrReplace('REAL_REGISTER_ENTERING_OR_LEAVING_DEFINED_RANGE ({0})'                      ,'{0}' , SINT_TO_STRING(Value));
  TriggerModeIo.REAL_REGISTER_ENTERING_OR_LEAVING_DEFINED_RANGE_INVERTED            : TRIGGER_MODE_IO_TO_STRING := StrReplace('REAL_REGISTER_ENTERING_OR_LEAVING_DEFINED_RANGE_INVERTED ({0})'             ,'{0}' , SINT_TO_STRING(Value));
ELSE
  TRIGGER_MODE_IO_TO_STRING := CONCAT('TRIGGER_MODE_IO_TO_STRING Function: Error -> no parsing for value ', SINT_TO_STRING(Value));
END_CASE
          
END_FUNCTION

FUNCTION TRIGGER_MODE_LIMIT_TO_STRING : STRING
// ------------------------------------------------------------------------- 
//  SRCI Robot Library                                                
// ------------------------------------------------------------------------- 
//                                                                           
//  Object:      TRIGGER_MODE_LIMIT_TO_STRING                                       
//  Author:      Thorsten Brach                                                
//  Date:        2025-03-02
//
//  Description:                                              
//   
//                                                                           
//  Copyright: 
//    (C) 2025 Thorsten Brach. All rights reserved                                                                                                                                            
//             Licensed under the MIT License.
//                                                                           
//  Disclaimer:                                                                           
//    This project is provided without any guarantee and can be used for   
//    private and commercial purposes. Any use is at the user’s 
//    own risk and responsibility.
//
// -------------------------------------------------------------------------
VAR_INPUT
  /// TriggerModeLimit
  Value : TriggerModeLimit;
END_VAR

            CASE Value 
OF
  TriggerModeLimit.INVALID         : TRIGGER_MODE_LIMIT_TO_STRING := StrReplace('INVALID ({0})'         ,'{0}' , SINT_TO_STRING(Value));
  TriggerModeLimit.JOINT_CURRENT   : TRIGGER_MODE_LIMIT_TO_STRING := StrReplace('JOINT_CURRENT ({0})'   ,'{0}' , SINT_TO_STRING(Value));
  TriggerModeLimit.FORCE           : TRIGGER_MODE_LIMIT_TO_STRING := StrReplace('FORCE ({0})'           ,'{0}' , SINT_TO_STRING(Value));
  TriggerModeLimit.FOLLOWING_ERROR : TRIGGER_MODE_LIMIT_TO_STRING := StrReplace('FOLLOWING_ERROR ({0})' ,'{0}' , SINT_TO_STRING(Value));
  TriggerModeLimit.TEMPERATURE     : TRIGGER_MODE_LIMIT_TO_STRING := StrReplace('TEMPERATURE ({0})'     ,'{0}' , SINT_TO_STRING(Value));
ELSE
  TRIGGER_MODE_LIMIT_TO_STRING := CONCAT('TRIGGER_MODE_LIMIT_TO_STRING Function: Error -> no parsing for value ', SINT_TO_STRING(Value));
END_CASE
          
END_FUNCTION

FUNCTION TRIGGER_MODE_MEASUREMENT_TO_STRING : STRING
// ------------------------------------------------------------------------- 
//  SRCI Robot Library                                                
// ------------------------------------------------------------------------- 
//                                                                           
//  Object:      TRIGGER_MODE_MEASUREMENT_TO_STRING                                       
//  Author:      Thorsten Brach                                                
//  Date:        2025-01-24
//
//  Description:                                              
//   
//                                                                           
//  Copyright: 
//    (C) 2025 Thorsten Brach. All rights reserved                                                                                                                                            
//             Licensed under the MIT License.
//                                                                           
//  Disclaimer:                                                                           
//    This project is provided without any guarantee and can be used for   
//    private and commercial purposes. Any use is at the user’s 
//    own risk and responsibility.
//
// -------------------------------------------------------------------------
VAR_INPUT
  /// TriggerMode
  Value : TriggerModeMeasurement;
END_VAR

            CASE Value 
OF
  TriggerModeMeasurement.NO_TRIGGER                   : TRIGGER_MODE_MEASUREMENT_TO_STRING := StrReplace('NO_TRIGGER ({0})'                   ,'{0}' , USINT_TO_STRING(Value));
  TriggerModeMeasurement.POSITIVE_START_NEGATIVE_STOP : TRIGGER_MODE_MEASUREMENT_TO_STRING := StrReplace('POSITIVE_START_NEGATIVE_STOP ({0})' ,'{0}' , USINT_TO_STRING(Value));
  TriggerModeMeasurement.POSITIVE_START_STOP          : TRIGGER_MODE_MEASUREMENT_TO_STRING := StrReplace('POSITIVE_START_STOP ({0})'          ,'{0}' , USINT_TO_STRING(Value));
ELSE
  TRIGGER_MODE_MEASUREMENT_TO_STRING := CONCAT('TRIGGER_MODE_MEASUREMENT_TO_STRING Function: Error -> no parsing for value ', USINT_TO_STRING(Value));
END_CASE
          
END_FUNCTION

FUNCTION TRIGGER_REACTION_MODE_TO_STRING : STRING
// ------------------------------------------------------------------------- 
//  SRCI Robot Library                                                
// ------------------------------------------------------------------------- 
//                                                                           
//  Object:      TRIGGER_REACTION_MODE_TO_STRING                                       
//  Author:      Thorsten Brach                                                
//  Date:        2025-02-01
//
//  Description:                                              
//   
//                                                                           
//  Copyright: 
//    (C) 2025 Thorsten Brach. All rights reserved                                                                                                                                            
//             Licensed under the MIT License.
//                                                                           
//  Disclaimer:                                                                           
//    This project is provided without any guarantee and can be used for   
//    private and commercial purposes. Any use is at the user’s 
//    own risk and responsibility.
//
// -------------------------------------------------------------------------
VAR_INPUT
  /// TriggerReactionMode
  Value : TriggerReactionMode;
END_VAR

            CASE Value 
OF

  TriggerReactionMode.NO_REACTION                : TRIGGER_REACTION_MODE_TO_STRING := StrReplace('NO_REACTION ({0})'                 ,'{0}' , SINT_TO_STRING(Value));
  TriggerReactionMode.INTERRUPT                  : TRIGGER_REACTION_MODE_TO_STRING := StrReplace('INTERRUPT ({0})'                   ,'{0}' , SINT_TO_STRING(Value));
  TriggerReactionMode.GROUP_STOP                 : TRIGGER_REACTION_MODE_TO_STRING := StrReplace('GROUP_STOP ({0})'                  ,'{0}' , SINT_TO_STRING(Value));
  TriggerReactionMode.DISABLE_ROBOT              : TRIGGER_REACTION_MODE_TO_STRING := StrReplace('DISABLE_ROBOT ({0})'               ,'{0}' , SINT_TO_STRING(Value));
  TriggerReactionMode.STOP_ACTUAL_MOTION_COMMAND : TRIGGER_REACTION_MODE_TO_STRING := StrReplace('STOP_ACTUAL_MOTION_COMMAND ({0})'  ,'{0}' , SINT_TO_STRING(Value));
ELSE
  TRIGGER_REACTION_MODE_TO_STRING := CONCAT('TRIGGER_REACTION_MODE_TO_STRING Function: Error -> no parsing for value ', SINT_TO_STRING(Value));
END_CASE
          
END_FUNCTION

FUNCTION TURN_MODE_TO_STRING : STRING
// ------------------------------------------------------------------------- 
//  SRCI Robot Library                                                
// ------------------------------------------------------------------------- 
//                                                                           
//  Object:      TURN_MODE_TO_STRING                                       
//  Author:      Thorsten Brach                                                
//  Date:        2025-01-23
//
//  Description:                                              
//   
//                                                                           
//  Copyright: 
//    (C) 2025 Thorsten Brach. All rights reserved                                                                                                                                            
//             Licensed under the MIT License.
//                                                                           
//  Disclaimer:                                                                           
//    This project is provided without any guarantee and can be used for   
//    private and commercial purposes. Any use is at the user’s 
//    own risk and responsibility.
//
// -------------------------------------------------------------------------
VAR_INPUT
  /// TurnMode
  Value : TurnMode;
END_VAR

            CASE Value 
OF
  TurnMode.USE_TURN_NUMBER : TURN_MODE_TO_STRING := StrReplace('USE_TURN_NUMBER ({0})','{0}' , USINT_TO_STRING(Value));
  TurnMode.SAME            : TURN_MODE_TO_STRING := StrReplace('SAME ({0})'           ,'{0}' , USINT_TO_STRING(Value));
  TurnMode.FREE            : TURN_MODE_TO_STRING := StrReplace('FREE ({0})'           ,'{0}' , USINT_TO_STRING(Value));
ELSE
  TURN_MODE_TO_STRING := CONCAT('TURN_MODE_TO_STRING Function: Error -> no parsing for value ', USINT_TO_STRING(Value));
END_CASE
          
END_FUNCTION

FUNCTION UNIT_LIMIT_AXIS_TO_STRING : STRING
// ------------------------------------------------------------------------- 
//  SRCI Robot Library                                                
// ------------------------------------------------------------------------- 
//                                                                           
//  Object:      ORI_MODE_TO_STRING                                       
//  Author:      Thorsten Brach                                                
//  Date:        2025-02-25
//
//  Description:                                              
//   
//                                                                           
//  Copyright: 
//    (C) 2025 Thorsten Brach. All rights reserved                                                                                                                                            
//             Licensed under the MIT License.
//                                                                           
//  Disclaimer:                                                                           
//    This project is provided without any guarantee and can be used for   
//    private and commercial purposes. Any use is at the user’s 
//    own risk and responsibility.
//
// -------------------------------------------------------------------------
VAR_INPUT
  /// UnitLimitAxis
  Value : UnitLimitAxis;
END_VAR

            CASE Value 
OF
  UnitLimitAxis.PERCENTAGE  : UNIT_LIMIT_AXIS_TO_STRING := StrReplace('PERCENTAGE ({0})'  ,'{0}' , USINT_TO_STRING(Value));
  UnitLimitAxis.NEWTONMETER : UNIT_LIMIT_AXIS_TO_STRING := StrReplace('NEWTONMETER ({0})' ,'{0}' , USINT_TO_STRING(Value));
  UnitLimitAxis.MILLIAMPERE : UNIT_LIMIT_AXIS_TO_STRING := StrReplace('MILLIAMPERE ({0})' ,'{0}' , USINT_TO_STRING(Value));
ELSE
  UNIT_LIMIT_AXIS_TO_STRING := CONCAT('UNIT_LIMIT_AXIS_TO_STRING Function: Error -> no parsing for value ', USINT_TO_STRING(Value));
END_CASE
          
END_FUNCTION

FUNCTION VALID_REAL_TO_STRING : STRING
// ------------------------------------------------------------------------- 
//  SRCI Robot Library                                                
// ------------------------------------------------------------------------- 
//                                                                           
//  Object:      VALID_REAL_TO_STRING                                       
//  Author:      Thorsten Brach                                                
//  Date:        2025-02-26
//
//  Description:                                              
//   
//                                                                           
//  Copyright: 
//    (C) 2025 Thorsten Brach. All rights reserved                                                                                                                                            
//             Licensed under the MIT License.
//                                                                           
//  Disclaimer:                                                                           
//    This project is provided without any guarantee and can be used for   
//    private and commercial purposes. Any use is at the user’s 
//    own risk and responsibility.
//
// -------------------------------------------------------------------------
VAR_INPUT
  /// Real
  Value : REAL;
END_VAR

            IF ( SysDepIsValidReal(Value))
THEN
  VALID_REAL_TO_STRING := REAL_TO_STRING(Value);
ELSE
  VALID_REAL_TO_STRING := 'NaN';
END_IF
          
END_FUNCTION

FUNCTION WORD_TO_STRING_BIN : STRING
// ------------------------------------------------------------------------- 
//  SRCI Robot Library                                                
// ------------------------------------------------------------------------- 
//                                                                           
//  Object:      WORD_TO_STRING_BIN                                       
//  Author:      Thorsten Brach                                                
//  Date:        2025-02-03
//
//  Description:                                              
//    Converts a BYTE to a STRING with binary notation  
//                                                                           
//  Copyright: 
//    (C) 2024 Thorsten Brach. All rights reserved                                                                                                                                            
//             Licensed under the MIT License.
//                                                                           
//  Disclaimer:                                                                           
//    This project is provided without any guarantee and can be used for   
//    private and commercial purposes. Any use is at the user’s 
//    own risk and responsibility.
//
// -------------------------------------------------------------------------
VAR_INPUT
 /// Value to convert
 Value : WORD; 
END_VAR

            WORD_TO_STRING_BIN := '2#';

IF (Value.15)
THEN
  WORD_TO_STRING_BIN := CONCAT(WORD_TO_STRING_BIN, '1');
ELSE
  WORD_TO_STRING_BIN := CONCAT(WORD_TO_STRING_BIN, '0');
END_IF

IF (Value.14)
THEN
  WORD_TO_STRING_BIN := CONCAT(WORD_TO_STRING_BIN, '1');
ELSE
  WORD_TO_STRING_BIN := CONCAT(WORD_TO_STRING_BIN, '0');
END_IF

IF (Value.13)
THEN
  WORD_TO_STRING_BIN := CONCAT(WORD_TO_STRING_BIN, '1');
ELSE
  WORD_TO_STRING_BIN := CONCAT(WORD_TO_STRING_BIN, '0');
END_IF

IF (Value.12)
THEN
  WORD_TO_STRING_BIN := CONCAT(WORD_TO_STRING_BIN, '1_');
ELSE
  WORD_TO_STRING_BIN := CONCAT(WORD_TO_STRING_BIN, '0_');
END_IF

IF (Value.11)
THEN
  WORD_TO_STRING_BIN := CONCAT(WORD_TO_STRING_BIN, '1');
ELSE
  WORD_TO_STRING_BIN := CONCAT(WORD_TO_STRING_BIN, '0');
END_IF

IF (Value.10)
THEN
  WORD_TO_STRING_BIN := CONCAT(WORD_TO_STRING_BIN, '1');
ELSE
  WORD_TO_STRING_BIN := CONCAT(WORD_TO_STRING_BIN, '0');
END_IF

IF (Value.09)
THEN
  WORD_TO_STRING_BIN := CONCAT(WORD_TO_STRING_BIN, '1');
ELSE
  WORD_TO_STRING_BIN := CONCAT(WORD_TO_STRING_BIN, '0');
END_IF

IF (Value.08)
THEN
  WORD_TO_STRING_BIN := CONCAT(WORD_TO_STRING_BIN, '1_');
ELSE
  WORD_TO_STRING_BIN := CONCAT(WORD_TO_STRING_BIN, '0_');
END_IF

IF (Value.7)
THEN
  WORD_TO_STRING_BIN := CONCAT(WORD_TO_STRING_BIN, '1');
ELSE
  WORD_TO_STRING_BIN := CONCAT(WORD_TO_STRING_BIN, '0');
END_IF

IF (Value.6)
THEN
  WORD_TO_STRING_BIN := CONCAT(WORD_TO_STRING_BIN, '1');
ELSE
  WORD_TO_STRING_BIN := CONCAT(WORD_TO_STRING_BIN, '0');
END_IF

IF (Value.5)
THEN
  WORD_TO_STRING_BIN := CONCAT(WORD_TO_STRING_BIN, '1');
ELSE
  WORD_TO_STRING_BIN := CONCAT(WORD_TO_STRING_BIN, '0');
END_IF

IF (Value.4)
THEN
  WORD_TO_STRING_BIN := CONCAT(WORD_TO_STRING_BIN, '1_');
ELSE
  WORD_TO_STRING_BIN := CONCAT(WORD_TO_STRING_BIN, '0_');
END_IF

IF (Value.3)
THEN
  WORD_TO_STRING_BIN := CONCAT(WORD_TO_STRING_BIN, '1');
ELSE
  WORD_TO_STRING_BIN := CONCAT(WORD_TO_STRING_BIN, '0');
END_IF

IF (Value.2)
THEN
  WORD_TO_STRING_BIN := CONCAT(WORD_TO_STRING_BIN, '1');
ELSE
  WORD_TO_STRING_BIN := CONCAT(WORD_TO_STRING_BIN, '0');
END_IF

IF (Value.1)
THEN
  WORD_TO_STRING_BIN := CONCAT(WORD_TO_STRING_BIN, '1');
ELSE
  WORD_TO_STRING_BIN := CONCAT(WORD_TO_STRING_BIN, '0');
END_IF


IF (Value.0)
THEN
  WORD_TO_STRING_BIN := CONCAT(WORD_TO_STRING_BIN, '1');
ELSE
  WORD_TO_STRING_BIN := CONCAT(WORD_TO_STRING_BIN, '0');
END_IF


WORD_TO_STRING_BIN := CONCAT(WORD_TO_STRING_BIN, ' (');
WORD_TO_STRING_BIN := CONCAT(WORD_TO_STRING_BIN, WORD_TO_STRING(Value));
WORD_TO_STRING_BIN := CONCAT(WORD_TO_STRING_BIN, ')');
          
END_FUNCTION

FUNCTION WORD_TO_STRING_HEX : STRING
// ------------------------------------------------------------------------- 
//  SRCI Robot Library                                                
// ------------------------------------------------------------------------- 
//                                                                           
//  Object:      WORD_TO_STRING_HEX                                       
//  Author:      Thorsten Brach                                                
//  Date:        2024-12-13
//
//  Description:                                              
//    Converts a WORD to a STRING with hex notation  
//                                                                           
//  Copyright: 
//    (C) 2024 Thorsten Brach. All rights reserved                                                                                                                                            
//             Licensed under the MIT License.
//                                                                           
//  Disclaimer:                                                                           
//    This project is provided without any guarantee and can be used for   
//    private and commercial purposes. Any use is at the user’s 
//    own risk and responsibility.
//
// -------------------------------------------------------------------------
VAR_INPUT
 /// Value to convert
 Value : WORD; 
END_VAR
VAR
  /// high Byte
 _highByte   : BYTE;      
  /// low Byte
 _lowByte    : BYTE;      
  /// high Nibble
 _highNibble : BYTE;     
  /// low Nibble 
 _lowNibble  : BYTE;     
  /// single Hex char
  hexChar    : STRING(1);
  /// Hex chars  
  hexChars   : ARRAY[0..15] OF STRING(1) := ['0', '1', '2', '3', '4', '5', '6', '7', '8', '9', 'A', 'B', 'C', 'D', 'E', 'F'];
END_VAR

            // get high and low byte from word
_highByte := WORD_TO_BYTE(SHR(Value, 8)); 
_lowByte  := WORD_TO_BYTE(Value AND 16#FF); 

// convert highest Byte to HEX
_highNibble := SHR(_highByte, 4);   
_lowNibble  := (_highByte AND 16#F);
WORD_TO_STRING_HEX := CONCAT(hexChars[_highNibble], hexChars[_lowNibble]);

// convert lowest Byte to HEX
_highNibble := SHR(_lowByte, 4); 
_lowNibble := _lowByte AND 16#F; 
WORD_TO_STRING_HEX := CONCAT(WORD_TO_STRING_HEX, CONCAT(hexChars[_highNibble], hexChars[_lowNibble]));

          
END_FUNCTION

FUNCTION WORK_AREA_REACTION_MODE_TO_STRING : STRING
// ------------------------------------------------------------------------- 
//  SRCI Robot Library                                                
// ------------------------------------------------------------------------- 
//                                                                           
//  Object:      WORK_AREA_REACTION_MODE_TO_STRING                                       
//  Author:      Thorsten Brach                                                
//  Date:        2025-02-01
//
//  Description:                                              
//   
//                                                                           
//  Copyright: 
//    (C) 2025 Thorsten Brach. All rights reserved                                                                                                                                            
//             Licensed under the MIT License.
//                                                                           
//  Disclaimer:                                                                           
//    This project is provided without any guarantee and can be used for   
//    private and commercial purposes. Any use is at the user’s 
//    own risk and responsibility.
//
// -------------------------------------------------------------------------
VAR_INPUT
  /// WorkAreaReactionMode
  Value : WorkAreaReactionMode;
END_VAR

            CASE Value 
OF
  WorkAreaReactionMode.NO_REACTION : WORK_AREA_REACTION_MODE_TO_STRING := StrReplace('NO_REACTION ({0})','{0}' , USINT_TO_STRING(Value));
  WorkAreaReactionMode.ABORT       : WORK_AREA_REACTION_MODE_TO_STRING := StrReplace('ABORT ({0})'      ,'{0}' , USINT_TO_STRING(Value));
  WorkAreaReactionMode.INTERRUPT   : WORK_AREA_REACTION_MODE_TO_STRING := StrReplace('INTERRUPT ({0})'  ,'{0}' , USINT_TO_STRING(Value));
ELSE
  WORK_AREA_REACTION_MODE_TO_STRING := CONCAT('WORK_AREA_REACTION_MODE_TO_STRING Function: Error -> no parsing for value ', USINT_TO_STRING(Value));
END_CASE
          
END_FUNCTION

/// Returns the given string, filled up on the right side to the given total length with the given substring
FUNCTION StrPadRight : STRING(255)
// ------------------------------------------------------------------------- 
//  SRCI Robot Library                                                
// ------------------------------------------------------------------------- 
//                                                                           
//  Object:      SwapBytes                                       
//  Author:      Thorsten Brach                                                
//  Date:        2024-12-18
//
//  Description:                                              
//   
//                                                                           
//  Copyright: 
//    (C) 2024 Thorsten Brach. All rights reserved                                                                                                                                            
//             Licensed under the MIT License.
//                                                                           
//  Disclaimer:                                                                           
//    This project is provided without any guarantee and can be used for   
//    private and commercial purposes. Any use is at the user’s 
//    own risk and responsibility.
//
// -------------------------------------------------------------------------
VAR_INPUT
  /// content string
  Str    : STRING(255);
  /// sub string
  SubStr : STRING(255);
  /// Length
  Length : INT; 
END_VAR

            WHILE(LEN(Str) < Length)
DO
 Str := CONCAT(Str, SubStr);
END_WHILE

StrPadRight := Str;
          
END_FUNCTION

/// Returns a given string where a given substing is replaced by another substring
FUNCTION StrReplace : STRING(255)
// ------------------------------------------------------------------------- 
//  SRCI Robot Library                                                
// ------------------------------------------------------------------------- 
//                                                                           
//  Object:      SwapBytes                                       
//  Author:      Thorsten Brach                                                
//  Date:        2024-12-18
//
//  Description:                                              
//   
//                                                                           
//  Copyright: 
//    (C) 2024 Thorsten Brach. All rights reserved                                                                                                                                            
//             Licensed under the MIT License.
//                                                                           
//  Disclaimer:                                                                           
//    This project is provided without any guarantee and can be used for   
//    private and commercial purposes. Any use is at the user’s 
//    own risk and responsibility.
//
// -------------------------------------------------------------------------
VAR_INPUT
  /// content string
  Str      : STRING(255);
  /// sub string with the old characters
  SubStr1  : STRING(255);
  /// sub string with the new characters
  SubStr2  : STRING(255);
END_VAR

            WHILE (FIND(Str, SubStr1) > 0)
DO  
  Str := Replace(Str, SubStr2, LEN(SubStr1), FIND(Str, SubStr1)); 
END_WHILE

StrReplace := Str;
          
END_FUNCTION

FUNCTION GetHalfeByteHi : BYTE
// ------------------------------------------------------------------------- 
//  SRCI Robot Library                                                
// ------------------------------------------------------------------------- 
//                                                                           
//  Object:      SwapBytes                                       
//  Author:      Thorsten Brach                                                
//  Date:        2024-12-18
//
//  Description:                                              
//   
//                                                                           
//  Copyright: 
//    (C) 2024 Thorsten Brach. All rights reserved                                                                                                                                            
//             Licensed under the MIT License.
//                                                                           
//  Disclaimer:                                                                           
//    This project is provided without any guarantee and can be used for   
//    private and commercial purposes. Any use is at the user’s 
//    own risk and responsibility.
//
// -------------------------------------------------------------------------
VAR_INPUT
  /// Increase payload pointer 
  Value : BYTE;
END_VAR

            GetHalfeByteHi.0 := Value.4;
GetHalfeByteHi.1 := Value.5;
GetHalfeByteHi.2 := Value.6;
GetHalfeByteHi.3 := Value.7;

          
END_FUNCTION

FUNCTION GetHalfeByteLo : BYTE
// ------------------------------------------------------------------------- 
//  SRCI Robot Library                                                
// ------------------------------------------------------------------------- 
//                                                                           
//  Object:      SwapBytes                                       
//  Author:      Thorsten Brach                                                
//  Date:        2024-12-18
//
//  Description:                                              
//   
//                                                                           
//  Copyright: 
//    (C) 2024 Thorsten Brach. All rights reserved                                                                                                                                            
//             Licensed under the MIT License.
//                                                                           
//  Disclaimer:                                                                           
//    This project is provided without any guarantee and can be used for   
//    private and commercial purposes. Any use is at the user’s 
//    own risk and responsibility.
//
// -------------------------------------------------------------------------
VAR_INPUT
  /// Increase payload pointer 
  Value : BYTE;
END_VAR

            GetHalfeByteLo.0 := Value.0;
GetHalfeByteLo.1 := Value.1;
GetHalfeByteLo.2 := Value.2;
GetHalfeByteLo.3 := Value.3;

          
END_FUNCTION

FUNCTION SwapBytes 
// ------------------------------------------------------------------------- 
//  SRCI Robot Library                                                
// ------------------------------------------------------------------------- 
//                                                                           
//  Object:      SwapBytes                                       
//  Author:      Thorsten Brach                                                
//  Date:        2024-06-01
//
//  Description:                                              
//   
//                                                                           
//  Copyright: 
//    (C) 2024 Thorsten Brach. All rights reserved                                                                                                                                            
//             Licensed under the MIT License.
//                                                                           
//  Disclaimer:                                                                           
//    This project is provided without any guarantee and can be used for   
//    private and commercial purposes. Any use is at the user’s 
//    own risk and responsibility.
//
// -------------------------------------------------------------------------
VAR_INPUT
  /// pointer to data type
  pValue : POINTER TO BYTE;
  /// size of data type
  Size  : UDINT;
END_VAR

VAR
  /// Pointer to low word low byte
  _pLwLb    : POINTER TO BYTE;
  /// Pointer to low word high byte
  _pLwHb    : POINTER TO BYTE;
  /// Pointer to high word low byte
  _pHwLb    : POINTER TO BYTE;
  /// Pointer to high word high byte
  _pHwHb    : POINTER TO BYTE;  
   /// temporary bytes
  _tmpBytes : ARRAY[1..4] OF BYTE;  
END_VAR

            IF ( RobotLibraryParameter.SWAP_BYTE_ORDER AND Size = 2)
THEN
 _pLwLb := pValue + 0;
 _pLwHb := pValue + 1;
  
  // swap bytes
 _tmpBytes[1] := _pLwHb^;
 _tmpBytes[2] := _pLwLb^;
  
  // copy bytes to data type
  SysDepMemCpy(pDest := pValue, pSrc := ADR(_tmpBytes), DataLen := Size);
END_IF


IF ( RobotLibraryParameter.SWAP_BYTE_ORDER AND Size = 4)
THEN
 _pLwLb := pValue + 0;
 _pLwHb := pValue + 1;
 _pHwLb := pValue + 2;
 _pHwHb := pValue + 3;
  
  // swap bytes
 _tmpBytes[1] := _pHwHb^;
 _tmpBytes[2] := _pHwLb^;
 _tmpBytes[3] := _pLwHb^;
 _tmpBytes[4] := _pLwLb^;
  
  // copy bytes to data type
  SysDepMemCpy( pDest := pValue, pSrc := ADR(_tmpBytes), DataLen := Size);  
END_IF
          
END_FUNCTION

FUNCTION SwapDword : DWORD
// ------------------------------------------------------------------------- 
//  SRCI Robot Library                                                
// ------------------------------------------------------------------------- 
//                                                                           
//  Object:      SwapDword                                       
//  Author:      Thorsten Brach                                                
//  Date:        2024-06-01
//
//  Description:                                              
//   
//                                                                           
//  Copyright: 
//    (C) 2024 Thorsten Brach. All rights reserved                                                                                                                                            
//             Licensed under the MIT License.
//                                                                           
//  Disclaimer:                                                                           
//    This project is provided without any guarantee and can be used for   
//    private and commercial purposes. Any use is at the user’s 
//    own risk and responsibility.
//
// -------------------------------------------------------------------------
VAR_INPUT
  /// Value
  Value : DWORD;
END_VAR

            SwapBytes(ADR(Value),SIZEOF(Value));

SwapDword := Value;
          
END_FUNCTION

FUNCTION SwapIecDate : IEC_DATE
// ------------------------------------------------------------------------- 
//  SRCI Robot Library                                                
// ------------------------------------------------------------------------- 
//                                                                           
//  Object:      SwapIecDate                                       
//  Author:      Thorsten Brach                                                
//  Date:        2024-06-09
//
//  Description:                                              
//   
//                                                                           
//  Copyright: 
//    (C) 2024 Thorsten Brach. All rights reserved                                                                                                                                            
//             Licensed under the MIT License.
//                                                                           
//  Disclaimer:                                                                           
//    This project is provided without any guarantee and can be used for   
//    private and commercial purposes. Any use is at the user’s 
//    own risk and responsibility.
//
// -------------------------------------------------------------------------
VAR_INPUT
  /// Value to swap
  Value : IEC_DATE;
END_VAR

            SwapBytes(ADR(Value),SIZEOF(Value));

SwapIecDate := Value;
          
END_FUNCTION

FUNCTION SwapIecTime : TOD
// ------------------------------------------------------------------------- 
//  SRCI Robot Library                                                
// ------------------------------------------------------------------------- 
//                                                                           
//  Object:      SwapTime                                       
//  Author:      Thorsten Brach                                                
//  Date:        2024-06-01
//
//  Description:                                              
//   
//                                                                           
//  Copyright: 
//    (C) 2024 Thorsten Brach. All rights reserved                                                                                                                                            
//             Licensed under the MIT License.
//                                                                           
//  Disclaimer:                                                                           
//    This project is provided without any guarantee and can be used for   
//    private and commercial purposes. Any use is at the user’s 
//    own risk and responsibility.
//
// -------------------------------------------------------------------------
VAR_INPUT
  /// Value
  Value : TOD;
END_VAR

            SwapBytes(ADR(Value),SIZEOF(Value));

SwapIecTime := Value;
          
END_FUNCTION

FUNCTION SwapInt : INT
// ------------------------------------------------------------------------- 
//  SRCI Robot Library                                                
// ------------------------------------------------------------------------- 
//                                                                           
//  Object:      SwapInt                                       
//  Author:      Thorsten Brach                                                
//  Date:        2024-06-01
//
//  Description:                                              
//   
//                                                                           
//  Copyright: 
//    (C) 2024 Thorsten Brach. All rights reserved                                                                                                                                            
//             Licensed under the MIT License.
//                                                                           
//  Disclaimer:                                                                           
//    This project is provided without any guarantee and can be used for   
//    private and commercial purposes. Any use is at the user’s 
//    own risk and responsibility.
//
// -------------------------------------------------------------------------
VAR_INPUT
  /// Value to swap
  Value : INT;
END_VAR

            SwapBytes(ADR(Value),SIZEOF(Value));

SwapInt := Value;
          
END_FUNCTION

FUNCTION SwapReal : REAL
// ------------------------------------------------------------------------- 
//  SRCI Robot Library                                                
// ------------------------------------------------------------------------- 
//                                                                           
//  Object:      SwapReal                                       
//  Author:      Thorsten Brach                                                
//  Date:        2024-06-01
//
//  Description:                                              
//   
//                                                                           
//  Copyright: 
//    (C) 2024 Thorsten Brach. All rights reserved                                                                                                                                            
//             Licensed under the MIT License.
//                                                                           
//  Disclaimer:                                                                           
//    This project is provided without any guarantee and can be used for   
//    private and commercial purposes. Any use is at the user’s 
//    own risk and responsibility.
//
// -------------------------------------------------------------------------
VAR_INPUT
  /// Value
  Value : REAL;
END_VAR

            SwapBytes(ADR(Value),SIZEOF(Value));

SwapReal := Value;
          
END_FUNCTION

FUNCTION SwapUdint : UDINT
// ------------------------------------------------------------------------- 
//  SRCI Robot Library                                                
// ------------------------------------------------------------------------- 
//                                                                           
//  Object:      SwapUdint                                       
//  Author:      Thorsten Brach                                                
//  Date:        2024-06-01
//
//  Description:                                              
//   
//                                                                           
//  Copyright: 
//    (C) 2024 Thorsten Brach. All rights reserved                                                                                                                                            
//             Licensed under the MIT License.
//                                                                           
//  Disclaimer:                                                                           
//    This project is provided without any guarantee and can be used for   
//    private and commercial purposes. Any use is at the user’s 
//    own risk and responsibility.
//
// -------------------------------------------------------------------------
VAR_INPUT
  /// Value
  Value : UDINT;
END_VAR

            SwapBytes(ADR(Value),SIZEOF(Value));

SwapUdint := Value;
          
END_FUNCTION

FUNCTION SwapUint : UINT
// ------------------------------------------------------------------------- 
//  SRCI Robot Library                                                
// ------------------------------------------------------------------------- 
//                                                                           
//  Object:      SwapUint                                       
//  Author:      Thorsten Brach                                                
//  Date:        2024-06-01
//
//  Description:                                              
//   
//                                                                           
//  Copyright: 
//    (C) 2024 Thorsten Brach. All rights reserved                                                                                                                                            
//             Licensed under the MIT License.
//                                                                           
//  Disclaimer:                                                                           
//    This project is provided without any guarantee and can be used for   
//    private and commercial purposes. Any use is at the user’s 
//    own risk and responsibility.
//
// -------------------------------------------------------------------------
VAR_INPUT
  /// Value to swap
  Value : UINT;
END_VAR

            SwapBytes(ADR(Value),SIZEOF(Value));

SwapUint := Value;
          
END_FUNCTION

FUNCTION SwapWord : WORD
// ------------------------------------------------------------------------- 
//  SRCI Robot Library                                                
// ------------------------------------------------------------------------- 
//                                                                           
//  Object:      SwapWord                                       
//  Author:      Thorsten Brach                                                
//  Date:        2024-06-01
//
//  Description:                                              
//   
//                                                                           
//  Copyright: 
//    (C) 2024 Thorsten Brach. All rights reserved                                                                                                                                            
//             Licensed under the MIT License.
//                                                                           
//  Disclaimer:                                                                           
//    This project is provided without any guarantee and can be used for   
//    private and commercial purposes. Any use is at the user’s 
//    own risk and responsibility.
//
// -------------------------------------------------------------------------
VAR_INPUT
  /// Value to swap
  Value : UINT;
END_VAR

            SwapBytes(ADR(Value),SIZEOF(Value));

SwapWord := Value;
          
END_FUNCTION

FUNCTION_BLOCK RobotLibraryBaseEnableFB EXTENDS RobotLibraryBaseFB
// ------------------------------------------------------------------------- 
//  SRCI Robot Library                                                
// ------------------------------------------------------------------------- 
//                                                                           
//  Object:      RobotLibraryBaseFB                                       
//  Author:      Thorsten Brach                                                
//  Date:        2024-08-11
//
//  Description:                                              
//   
//                                                                           
//  Copyright: 
//    (C) 2024 Thorsten Brach. All rights reserved                                                                                                                                            
//             Licensed under the MIT License.
//                                                                           
//  Disclaimer:                                                                           
//    This project is provided without any guarantee and can be used for   
//    private and commercial purposes. Any use is at the user’s 
//    own risk and responsibility.
//
// -------------------------------------------------------------------------
VAR_INPUT
  /// Set TRUE to activate / Set False to deactivate
  Enable            : BOOL;
END_VAR

VAR_OUTPUT
  /// FB is being processed
  Busy              : BOOL;
  /// TRUE while function is active
  Enabled           : BOOL;
END_VAR

VAR
  /// Rising edge for enable
  {attribute 'hide'}
 _enable_R          : R_TRIG;
  /// Falling edge for enable
  {attribute 'hide'}
 _enable_F          : F_TRIG;
END_VAR

            SUPER^(AxesGroup := AxesGroup);
          

METHOD PROTECTED OnCall
VAR_IN_OUT
  /// Robot assignment of function
  AxesGroup : AxesGroup; 
END_VAR

VAR
  /// internal return value
 _retVal : DINT;
END_VAR
                  SUPER^.OnCall(AxesGroup := AxesGroup);

// building rising and falling edges
_enable_R( CLK := Enable);
_enable_F( CLK := Enable);


// Check command execution is allowed ?
IF ((     Enable                                 ) AND
    ( NOT AxesGroup.State.Initialized            ) AND
    ( NOT AxesGroup.State.Synchronized           ) AND
    (     MyType <> 'MC_ExchangeConfigurationFB' ) AND // is part of init sequence
    (     MyType <> 'MC_ReadMessagesFB'          ) AND // is part of init sequence
    (     MyType <> 'MC_ReadRobotDataFB'         ))    // is part of init sequence
THEN
  SetError( ErrorID := RobotLibraryErrorIdEnum.ERR_COMMANDS_NOT_ENABLED, Overwrite := TRUE );
  Error   := TRUE;
  Busy    := FALSE; 
END_IF


// On execution started
IF ( _enable_R.Q )
THEN
  OnExecStart(AxesGroup := AxesGroup);
END_IF


// On execution cancel  
IF ( Busy ) AND ( _enable_F.Q ) 
THEN
  // set cancel flag
 _cancel := TRUE;
END_IF

IF ( _cancel )
THEN
  // call Cancel
 _retVal := OnExecCancel(AxesGroup := AxesGroup);
  
  // done or error ?
  IF ( _retVal <> RobotLibraryConstants.RUNNING )
  THEN
    // reset cancel flag
   _cancel := FALSE;
	END_IF
END_IF


// On execution error clear
IF ( Error ) AND ( _enable_F.Q )
THEN
  // set ClearError flag
 _clearError := TRUE;
END_IF

IF ( _clearError )
THEN
 _retVal := OnExecErrorClear(AxesGroup := AxesGroup); 

  // done or error ?
  IF ( _retVal <> RobotLibraryConstants.RUNNING )
  THEN
    // reset ClearError flag
   _clearError := FALSE;
	END_IF
END_IF
                
END_METHOD

METHOD Protected OnExecCancel : DINT
VAR_IN_OUT
  /// Robot assignment of function
  AxesGroup : AxesGroup; 
END_VAR
VAR
  /// internal return value 
 _retVal    : DINT;
END_VAR
                  OnExecCancel := Reset();

// Create log entry
CreateLogMessagePara1 ( Timestamp   := AxesGroup.State.SystemTime,
                        MessageType := MessageType.CMD,
                        Severity    := Severity.DEBUG,
                        MessageCode := 0,
                        MessageText := 'Execution of {1} cancled ',
                        Para1       := MyType);                 

// try to remove cmd
_retVal := AxesGroup.Acyclic.ActiveCommandRegister.RemoveCmd(_uniqueID);

IF (_retVal = RobotLibraryConstants.OK)
THEN
  // Create log entry
  CreateLogMessagePara1 ( Timestamp   := AxesGroup.State.SystemTime,
                          MessageType := MessageType.CMD,
                          Severity    := Severity.DEBUG,
                          MessageCode := 0,
                          MessageText := '{1} successfully removed from ACR',
                          Para1       := MyType);                 
ELSE
  // Create log entry
  CreateLogMessagePara1 ( Timestamp   := AxesGroup.State.SystemTime,
                          MessageType := MessageType.CMD,
                          Severity    := Severity.DEBUG,
                          MessageCode := 0,
                          MessageText := '{1} was not removed from ACR because execution was already in progress',
                          Para1       := MyType);                 
END_IF   
                
END_METHOD

METHOD PROTECTED OnExecErrorClear : DINT
VAR_IN_OUT
  /// Robot assignment of function
  AxesGroup : AxesGroup; 
END_VAR
                  OnExecErrorClear := RobotLibraryConstants.RUNNING;

CASE _stepClearError OF
  
  0:  // Reset 
      Reset();
      // trigger parameter update to disable FB
     _parameterUpdateInternal := TRUE;
      // call Check Parameter changed method to trigger the parameter update to deactivate jogging mode
      CheckParameterChanged(AxesGroup := AxesGroup);
      // set timeout
      SetTimeout(PT := _timeoutClearError, rTimer := _timerClearError);
      // inc step counter
     _stepClearError := _stepClearError + 1; 
      
  1: IF ( _responseReceived )
     THEN     
       // reset response received flag
      _responseReceived := FALSE;
       // reset step counter
      _stepClearError := 0;
       // finished
       OnExecErrorClear := RobotLibraryConstants.OK;
     ELSE
       // timeout exceeded ? 
       IF (CheckTimeout(_timerClearError) = RobotLibraryConstants.OK)
       THEN
         OnExecErrorClear := RobotLibraryConstants.HAS_ERROR;
       END_IF
	   END_IF
ELSE
  // invalid step
  SetError( ErrorID := RobotLibraryErrorIdEnum.ERR_INVALID_STEP, Overwrite := TRUE );
END_CASE


// reset step counter
IF (OnExecErrorClear <> RobotLibraryConstants.RUNNING)
THEN
 _stepClearError := 0;
END_IF
                
END_METHOD

METHOD PROTECTED OnExecRun : DINT
VAR_IN_OUT
  /// Robot assignment of function
  AxesGroup : AxesGroup; 
END_VAR
                  
                
END_METHOD

METHOD PROTECTED OnExecStart : DINT
VAR_IN_OUT
  /// Robot assignment of function
  AxesGroup : AxesGroup; 
END_VAR
                  
                
END_METHOD

METHOD PROTECTED OnUpdateStateFlags
VAR_INPUT
  /// Command message state
  State : CmdMessageState;
END_VAR
                  CASE State OF

  // No operation or process is active
  CmdMessageState.EMPTY               :;
  // Created but not yet started
  CmdMessageState.CREATED             :;
  // Buffered and awaiting execution
  CmdMessageState.BUFFERED            :;
  // Buffered in planner for future execution
  CmdMessageState.BUFFERED_IN_PLANNER :;
  // Currently active and in progress
  CmdMessageState.ACTIVE              :;
  // Interrupted and awaiting continuation
  CmdMessageState.INTERRUPTED         :;
  // Requested for abort
  CmdMessageState.ABORT_REQUEST       :;
  // Successfully completed
  CmdMessageState.DONE                : Busy := FALSE;
  // Aborted before completion
  CmdMessageState.ABORTED             : Busy := FALSE;
  // Encountered an error during execution
  CmdMessageState.ERROR               : Busy := FALSE;
END_CASE
                
END_METHOD

METHOD PROTECTED Reset : DINT
VAR_INPUT
END_VAR
                  Reset := SUPER^.Reset();

Busy    := FALSE;
Enabled := FALSE;
                
END_METHOD
END_FUNCTION_BLOCK

FUNCTION_BLOCK RobotLibraryBaseExecuteFB EXTENDS RobotLibraryBaseFB
// ------------------------------------------------------------------------- 
//  SRCI Robot Library                                                
// ------------------------------------------------------------------------- 
//                                                                           
//  Object:      RobotLibraryBaseFB                                       
//  Author:      Thorsten Brach                                                
//  Date:        2024-08-11
//
//  Description:                                              
//   
//                                                                           
//  Copyright: 
//    (C) 2024 Thorsten Brach. All rights reserved                                                                                                                                            
//             Licensed under the MIT License.
//                                                                           
//  Disclaimer:                                                                           
//    This project is provided without any guarantee and can be used for   
//    private and commercial purposes. Any use is at the user’s 
//    own risk and responsibility.
//
// -------------------------------------------------------------------------
VAR_INPUT
  /// Start of the command at the rising edge
  Execute         : BOOL;
END_VAR
VAR_OUTPUT
  /// The command has been completed successfully
  Done            : BOOL;
  /// FB is being processed
  Busy            : BOOL;
  /// Command is transferred and confirmed by the RC
//  CommandBuffered : BOOL;  
END_VAR


VAR
  /// Rising edge for execute
  {attribute 'hide'}
 _execute_R       : R_TRIG;
  /// Falling edge for execute
  {attribute 'hide'}
 _execute_F       : F_TRIG;
END_VAR

            SUPER^(AxesGroup := AxesGroup);
          

// Base implementation must be called ! 
METHOD PROTECTED OnCall
VAR_IN_OUT
  /// Robot assignment of function
  AxesGroup         : AxesGroup; 
END_VAR

VAR
  /// internal return value
 _retVal : DINT;
END_VAR
                  SUPER^.OnCall(AxesGroup := AxesGroup);

// building rising and falling edges
_execute_R( CLK := Execute);
_execute_F( CLK := Execute);


// Check command execution is allowed ?
IF ((     Execute                                ) AND
    ( NOT AxesGroup.State.CMDsEnabled            ) AND
    (     MyType <> 'MC_ExchangeConfigurationFB' ) AND // is part of init sequence
    (     MyType <> 'MC_ReadMessagesFB'          ) AND // is part of init sequence
    (     MyType <> 'MC_ReadRobotDataFB'         ))    // is part of init sequence
THEN
  SetError( ErrorID := RobotLibraryErrorIdEnum.ERR_COMMANDS_NOT_ENABLED, Overwrite := TRUE );
  Error   := TRUE;
  Busy    := FALSE;
END_IF


// On execution started
IF ( _execute_R.Q )
THEN
  OnExecStart(AxesGroup := AxesGroup);
END_IF


// On execution cancel  
IF ( Busy ) AND ( _execute_F.Q ) 
THEN
  // set cancel flag
 _cancel := TRUE;
END_IF

IF ( _cancel )
THEN
  // call Cancel
 _retVal := OnExecCancel(AxesGroup := AxesGroup);
  
  // done or error ?
  IF ( _retVal <> RobotLibraryConstants.RUNNING )
  THEN
    // reset cancel flag
   _cancel := FALSE;
	END_IF
END_IF


// On execution error clear
IF ( Error ) AND ( _execute_F.Q )
THEN
  // set ClearError flag
 _clearError := TRUE;
END_IF

IF ( _clearError )
THEN
 _retVal := OnExecErrorClear(AxesGroup := AxesGroup); 

  // done or error ?
  IF ( _retVal <> RobotLibraryConstants.RUNNING )
  THEN
    // reset ClearError flag
   _clearError := FALSE;
	END_IF
END_IF
                
END_METHOD

METHOD PROTECTED OnExecCancel : DINT
VAR_IN_OUT
  /// Robot assignment of function
  AxesGroup : AxesGroup; 
END_VAR
VAR
  /// internal return value 
 _retVal    : DINT;
END_VAR
                  // Create log entry
CreateLogMessagePara1 ( Timestamp   := AxesGroup.State.SystemTime,
                        MessageType := MessageType.CMD,
                        Severity    := Severity.DEBUG,
                        MessageCode := 0,
                        MessageText := 'Execution of {1} cancled ',
                        Para1       := MyType);                 

// try to remove cmd
_retVal := AxesGroup.Acyclic.ActiveCommandRegister.RemoveCmd(_uniqueID);


IF (_retVal = RobotLibraryConstants.OK)
THEN
  // Create log entry
  CreateLogMessagePara1 ( Timestamp   := AxesGroup.State.SystemTime,
                          MessageType := MessageType.CMD,
                          Severity    := Severity.DEBUG,
                          MessageCode := 0,
                          MessageText := '{1} successfully removed from ACR',
                          Para1       := MyType);                 
ELSE
  // Create log entry
  CreateLogMessagePara1 ( Timestamp   := AxesGroup.State.SystemTime,
                          MessageType := MessageType.CMD,
                          Severity    := Severity.DEBUG,
                          MessageCode := 0,
                          MessageText := '{1} was not removed from ACR because execution was already in progress',
                          Para1       := MyType);                 
END_IF


OnExecCancel := Reset();     
                
END_METHOD

